PROGRAM P_ComEL6001
VAR
	fbEL6001Ctrl		: SerialLineControl;
	bEL6001CtrlError	: BOOL;
	eEL6001CtrlErrorID	: ComError_t;
END_VAR

//***********************************************************************************
//
// ETH Zürich / Robotic Fabrication Lab
// HIB C 13 / Stefano-Franscini-Platz 1
// CH-8093 Zürich
// 
// ***********************************************************************************
// 
// PROJECT     :  ?? 
// 
// FUNCTION    :  Communication with EL6001 (RS-232)
// 
// AUTHOR      :  Mathias Suter
// 
// EMAIL       :  mathias.suter@solinaut.ch
// 
// Copyright   :  ETH Zürich (CH) 2021
//
// ***********************************************************************************


//
// Communication with EL6001
fbEL6001Ctrl(
	Mode:= SERIALLINEMODE_EL6_22B, 
	pComIn:= ADR(GVL.stIn_EL6001), 
	pComOut:= ADR(GVL.stOut_EL6001), 
	SizeComIn:= UINT_TO_INT(SIZEOF(GVL.stIn_EL6001)), 
	Error=> , 
	ErrorID=> , 
	TxBuffer:= GVL.TxBufferEL, 
	RxBuffer:= GVL.RxBufferEL );
		
//
// Output ErrorID, if Error detected
IF fbEL6001Ctrl.Error THEN
	bEL6001CtrlError := TRUE;
	eEL6001CtrlErrorID := fbEL6001Ctrl.ErrorID;
END_IF

END_PROGRAM

(* stored: Version 1.1.0.1, ProductVersion 3.1.4024.11
   POU P_ComEL6001: Id {9a20473f-0d3f-4584-b429-33e10587a848}, SpecialFunc None *)
